% RSLogix 500 project AUTOMATIC TRAIN COMPARTMENT WASHING SYSTEM.RSS, saved by version 8.30.00.16 %
PROJECT "UNTITLED"    % processor: Bul.1763 MicroLogix 1100 Series B %

PROGRAM FILES
  LAD 2   7 rungs

DATA FILES
  O0 OUTPUT  4 elements
  I1 INPUT  6 elements
  S2 STATUS  66 elements
  B3 BINARY  1 elements
  T4 TIMER  1 elements
  C5 COUNTER  1 elements
  R6 CONTROL  1 elements
  N7 INTEGER  1 elements
  F8 FLOAT  1 elements

LADDER 2
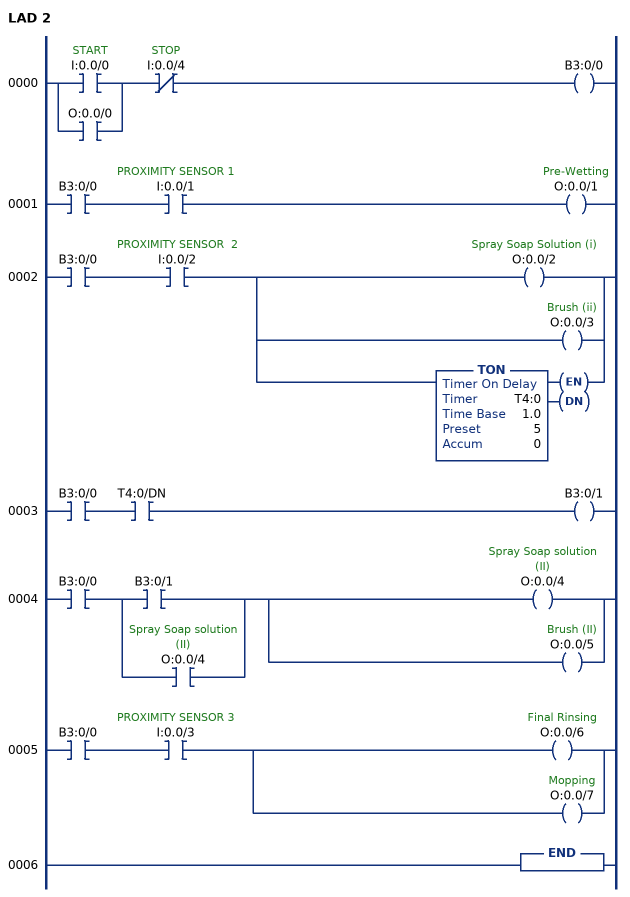
% Rung: 0 %
SOR BST XIC I:0.0/0 NXB XIC O:0.0/0 BND XIO I:0.0/4 OTE B3:0/0 EOR
%   I:0.0/0  "START" %
%   I:0.0/4  "STOP" %
% Rung: 1 %
SOR XIC B3:0/0 XIC I:0.0/1 OTE O:0.0/1 EOR
%   I:0.0/1  "PROXIMITY SENSOR 1" %
%   O:0.0/1  "Pre-Wetting" %
% Rung: 2 %
SOR XIC B3:0/0 XIC I:0.0/2 BST OTE O:0.0/2 NXB OTE O:0.0/3 NXB TON T4:0 1.0 5 0 BND EOR
%   I:0.0/2  "PROXIMITY SENSOR  2" %
%   O:0.0/2  "Spray Soap Solution (i)" %
%   O:0.0/3  "Brush (ii)" %
% Rung: 3 %
SOR XIC B3:0/0 XIC T4:0/DN OTE B3:0/1 EOR
% Rung: 4 %
SOR XIC B3:0/0 BST XIC B3:0/1 NXB XIC O:0.0/4 BND BST OTE O:0.0/4 NXB OTE O:0.0/5 BND EOR
%   O:0.0/4  "Spray Soap solution (II)" %
%   O:0.0/5  "Brush (II)" %
% Rung: 5 %
SOR XIC B3:0/0 XIC I:0.0/3 BST OTE O:0.0/6 NXB OTE O:0.0/7 BND EOR
%   I:0.0/3  "PROXIMITY SENSOR 3" %
%   O:0.0/6  "Final Rinsing" %
%   O:0.0/7  "Mopping" %
% Rung: 6 %
SOR END EOR

DATA TABLE (non-zero values as saved)
DATA T4
% .PRE .ACC %
% T4:0 % 5 0
